# B&R Automation Studio project Software_lab_3
Automation Studio 4.5.2.102

## Logical view

Binary libraries used (declarations not repeated): operator, runtime, astime, AsIecCon, AsBrStr, brsystem, sys_lib, AsIOTime, standard, asstring, Acp10_MC, Acp10man, NcGlobal, Acp10par, Acp10sim, Acp10sdc

### Global.var - Global variables
```iecst
VAR
	Axis_X : ACP10AXIS_typ;
	Axis_X_HW : SdcHwCfg_typ := (0);
	Axis_X_DrvIf : SdcDrvIf16_typ := (0);
	Axis_X_EncIf : SdcEncIf16_typ;
	Axis_X_DiDoIf : SdcDiDoIf_typ := (0);
	Axis_X_ModuleOk : BOOL := 0;
END_VAR
```

### Package Logical/Libraries - Global libraries

### Library Logical/Libraries/MotorCtrl (ANSIC)

#### MotorCtrl.fun - Exported functions and function blocks
```iecst
FUNCTION_BLOCK FB_Regulator
	VAR_INPUT
		e : REAL;
		e_prev : REAL;
	END_VAR
	VAR_OUTPUT
		u : REAL;
	END_VAR
	VAR
		u_raw : REAL;
		k_p : REAL;
		k_i : REAL;
		integrator : FB_Integrator;
		iyOld : REAL;
		max_abs_value : REAL;
	END_VAR
END_FUNCTION_BLOCK

FUNCTION_BLOCK FB_Motor
	VAR_INPUT
		u : REAL;
	END_VAR
	VAR_OUTPUT
		w : REAL;
		phi : REAL;
	END_VAR
	VAR
		integrator : FB_Integrator;
		integrator_phi : FB_Integrator;
		Tm : REAL;
		ke : REAL;
		enable_reg : BOOL;
	END_VAR
END_FUNCTION_BLOCK

FUNCTION_BLOCK FB_Integrator
	VAR_INPUT
		in : REAL;
	END_VAR
	VAR_OUTPUT
		out : REAL;
	END_VAR
	VAR
		dt : REAL;
		direct : BOOL;
	END_VAR
END_FUNCTION_BLOCK

FUNCTION_BLOCK FB_Axis
	VAR_INPUT
		u : USINT;
		endswitch_a_reached : BOOL;
		endswitch_b_reached : BOOL;
	END_VAR
	VAR_OUTPUT
		reset_error : BOOL;
		reset_counter : BOOL;
		pwm_value : INT;
		counter : INT;
		speed : REAL;
	END_VAR
	VAR
		last_counter : INT;
		InMotion : BOOL;
	END_VAR
END_FUNCTION_BLOCK
```

#### FB_Regulator.c
```c
#include <bur/plctypes.h>
#ifdef __cplusplus
	extern "C"
	{
#endif
#include "MotorCtrl.h"
#ifdef __cplusplus
	};
#endif
/* TODO: Add your comment here */
void FB_Regulator(struct FB_Regulator* inst)
{
	if (inst->integrator.direct)
		inst->integrator.in = inst->k_i * inst->e_prev + inst->iyOld / inst->integrator.dt;
	else
		inst->integrator.in = inst->k_i * inst->e + inst->iyOld / inst->integrator.dt;
	FB_Integrator(&inst->integrator);
	inst->u_raw = (inst->k_p * inst->e <= inst->max_abs_value ? inst->k_p * inst->e : inst->max_abs_value) +
		inst->integrator.out;
	inst->u = inst->u_raw < inst->max_abs_value ? inst->u_raw : inst->max_abs_value;
	inst->iyOld = inst->u - inst->u_raw;
}
```

#### FB_Motor.c
```c
#include <bur/plctypes.h>
#ifdef __cplusplus
	extern "C"
	{
#endif
#include "MotorCtrl.h"
#ifdef __cplusplus
	};
#endif
/* TODO: Add your comment here */
void FB_Motor(struct FB_Motor* inst)
{
	inst->integrator.in = (inst->u / inst->ke - inst->w) / inst->Tm;
	FB_Integrator(&inst->integrator);
	inst->w = inst->integrator.out;

	inst->integrator_phi.in = inst->w;
	FB_Integrator(&inst->integrator_phi);
	inst->phi = inst->integrator_phi.out;
}
```

#### FB_Axis.c
```c
#include <bur/plctypes.h>
#ifdef __cplusplus
	extern "C"
	{
#endif
#include "MotorCtrl.h"
#ifdef __cplusplus
	};
#endif
/* TODO: Add your comment here */
void FB_Axis(struct FB_Axis* inst)
{
	if (inst->InMotion)
	{
		if (inst->endswitch_a_reached || inst->endswitch_b_reached)
		{
			inst->pwm_value = 0;
			inst->speed = 0;
			inst->reset_error = 1;
			inst->InMotion = 0;
		}
		else
		{
			inst->pwm_value = inst->u / 24.0 * 32767;
			inst->speed = 50;
			inst->reset_error = 0;
		}
	}
}
```

### Program Logical/SDCAxisCtrlX (ANSIC)

#### Variables.var
```iecst
VAR
	axis_X : FB_Axis;
	coil_powered : BOOL;
	coil_pwm_value : INT;
	fb_regulator : FB_Regulator;
	pwm_period : UINT;
	min_task : INT := 7000;
END_VAR
```

#### Main.c
```c
/*#include <bur/plctypes.h>
#include <math.h>

#ifdef _DEFAULT_INCLUDES
	#include <AsDefault.h>
#endif

#define MOTORS_COUNT 3

void _INIT MainINIT(void)
{
	//Устанавливаем типы SDC модулей
	Axis_X_HW.EncIf1_Typ = ncSDC_ENC16;
	Axis_X_HW.DiDoIf_Typ = ncSDC_DIDO;
	Axis_X_HW.DrvIf_Typ = ncSDC_DRVSERVO16;
	//Устанавливаем имена переменных
	strcpy(Axis_X_HW.EncIf1_Name, "Axis_X_EncIf");
	strcpy(Axis_X_HW.DrvIf_Name, "Axis_X_DrvIf");
	strcpy(Axis_X_HW.DiDoIf_Name, "Axis_X_DiDoIf");
	//Устанавливаем входы готовности и нормальной
	работы
	Axis_X_EncIf.iEncOK = 1;
	Axis_X_DrvIf.iDrvOK = 1;
	Axis_X_DrvIf.iStatusEnable = 1;
	Axis_X_DiDoIf.iDriveReady = 1;

	Axis_X_EncIf.iLifeCnt++;
	Axis_X_DiDoIf.iLifeCntDriveEnable++;
	Axis_X_DiDoIf.iLifeCntDriveReady++;
	Axis_X_DiDoIf.iLifeCntNegHwEnd++;
	Axis_X_DiDoIf.iLifeCntPosHwEnd++;
	Axis_X_DiDoIf.iLifeCntReference++;
	Axis_X_DrvIf.iLifeCnt++;
	Axis_X_EncIf.iActTime = (INT)AsIOTimeCyclicStart();

	int i = 0;
	for (; i < MOTORS_COUNT; i++)
	{
		motors[i].pwm_value = 0;
		motors[i].pwm_percentage = 0;
		motors[i].counter = 0;
		motors[i].coordinate = 0;
		motors[i].button_status = 0;
		motors[i].reset_error = 0;
		motors[i].endswitch_a_reached = 0;
		motors[i].endswitch_b_reached = 0;
	}
	pwm_period = 200;
	coil_powered = 0;
	coil_pwm_value = 0;
	emergency_stop = 0;
	current_motor_index = 0;

	check = 0;
	a = 0;
	n = 0;
}

void _CYCLIC MainCYCLIC(void)
{
	int i = 0, j = 0;
	if (emergency_stop)  //аварийная остановка
	{
		for (i = 0; i < MOTORS_COUNT; i++)
		{
			motors[i].pwm_value = 0;
			motors[i].pwm_percentage = 0;
		}
		coil_powered = 0;
		check = 0;
		emergency_stop = 0;
	}
	current_motor = &motors[current_motor_index];
	for (i = 0; i < MOTORS_COUNT; i++)  //цикл для обозначения на экране текущей степени (кнопка подсвечивается белым цветом)
	{
		MotorFunctionBlock(&motors[i]);
		if (current_motor == &motors[i])
		{
			motors[i].button_status = 1 << 1;
		}
		else
		{
			motors[i].button_status = 0;
		}
	}
	if (coil_powered)  //проверяем напряжение на катушке
	{
		coil_pwm_value = 32767;
		if (check)
		{
			switch (mode)  //проверяем выбранный режим
			{
				case 1:
					switch (path)  //проверяем выбранный контур, разбиваем его и заполняем массив координат соответствующими значениями
					{
						case 1:
							for (i = 0; i < 20; i++)
							{
								coordX[i] = 150 * pi * i / (10*sqrt(2));
								coordY[i] = 150 * pi * i / (10*sqrt(2));
								coordZ[i] = 250 * sin(sqrt(coordX[i] * coordX[i] + coordY[i] * coordY[i]) / 150);
							}
							break;
						case 2:
							for (i = 0; i < 20; i++)
							{
								coordX[i] = 30 * i;
								coordY[i] = 30 * i;
								coordZ[i] = (coordX[i] * coordX[i] + coordY[i] * coordY[i]) / 180;
							}
							break;
						case 0:
							break;
					}
					distX = coordX[a+1] - coordX[a];  //длина полученных отрезков
					distY = coordY[a+1] - coordY[a];
					distZ = coordZ[a+1] - coordZ[a];
					if ((fabs(distX) >= fabs(distY)) && (fabs(distX) >= fabs(distZ)))  //поиск наибольшей проекции каждого отрезка
					{
						index[a] = 2;
					}
					if ((fabs(distY) >= fabs(distX)) && (fabs(distY) >= fabs(distZ)))
					{
						index[a] = 0;
					}
					if ((fabs(distZ) >= fabs(distX)) && (fabs(distZ) >= fabs(distY)))
					{
						index[a] = 1;
					}
					if (index[a] == 2)  //проекция на ось X наибольшая
					{
						if (motors[2].counter > coordX[a+1])  //если степень находится за следующей точкой, то двигаем её в обратном направлении
						{
							motors[2].pwm_percentage_float = -50.0;
						}
						if (motors[2].counter < coordX[a+1])  //если перед точкой, то в прямом направлении
						{
							motors[2].pwm_percentage_float = 50.0;
						}
						motors[0].pwm_percentage_float = (distY * motors[2].pwm_percentage_float) / distX;  //вычисляем реальное значение ШИМ (в процентах)
						motors[1].pwm_percentage_float = (distZ * motors[2].pwm_percentage_float) / distX;
						if ((motors[2].counter >= (coordX[a+1] - 2)) && (motors[2].counter <= (coordX[a+1] + 2)))
						{
							if (a < 18)  //проверка пройденных точек
							{
								a++;
							}
							else  //если все точки пройдены, то отключаем степени и сбрасываем выбранные режим и контур
							{
								for (i = 0; i < MOTORS_COUNT; i++)
								{
									motors[i].pwm_percentage_float = 0.0;
									motors[i].pwm_value_float = 0.0;
									motors[i].pwm_percentage = 0;
									motors[i].pwm_value = 0;
								}
								check = 0;
								mode = 0;
								path = 0;
								a = 0;
							}
						}
					}
					if (index[a] == 0)  //проекция на ось Y максимальная
					{
						if (motors[0].counter > coordY[a+1])  //если степень находится за следующей точкой, то двигаем её в обратном направлении
						{
							motors[0].pwm_percentage_float = -50.0;
						}
						if (motors[0].counter < coordY[a+1])  //если перед точкой, то в прямом направлении
						{
							motors[0].pwm_percentage_float = 50.0;
						}
						motors[2].pwm_percentage_float = (distX * motors[0].pwm_percentage_float) / distY;  //вычисляем реальное значение ШИМ (в процентах)
						motors[1].pwm_percentage_float = (distZ * motors[0].pwm_percentage_float) / distY;
						if ((motors[0].counter >= (coordY[a+1] - 2)) && (motors[0].counter <= (coordY[a+1] + 2)))
						{
							if (a < 18)  //проверка пройденных точек
							{
								a++;
							}
							else  //если все точки пройдены, то отключаем степени и сбрасываем выбранные режим и контур
							{
								for (i = 0; i < MOTORS_COUNT; i++)
								{
									motors[i].pwm_percentage_float = 0.0;
									motors[i].pwm_value_float = 0.0;
									motors[i].pwm_percentage = 0;
									motors[i].pwm_value = 0;
								}
								check = 0;
								mode = 0;
								path = 0;
								a = 0;
							}
						}
					}
					if (index[a] == 1)  //проекция на ось Z максимальная
					{
						if (motors[1].counter > coordZ[a+1])  //если степень находится за следующей точкой, то двигаем её в обратном направлении
						{
							motors[1].pwm_percentage_float = -50.0;
						}
						if (motors[1].counter < coordZ[a+1])  //если перед точкой, то в прямом направлении
						{
							motors[1].pwm_percentage_float = 50.0;
						}
						motors[2].pwm_percentage_float = (distX * motors[1].pwm_percentage_float) / distZ;  //вычисляем реальное значение ШИМ (в процентах)
						motors[0].pwm_percentage_float = (distY * motors[1].pwm_percentage_float) / distZ;
						if ((motors[1].counter >= (coordZ[a+1] - 2)) && (motors[1].counter <= (coordZ[a+1] + 2)))
						{
							if (a < 18)  //проверка пройденных точек
							{
								a++;
							}
							else  //если все точки пройдены, то отключаем степени и сбрасываем выбранные режим и контур
							{
								for (i = 0; i < MOTORS_COUNT; i++)
								{
									motors[i].pwm_percentage_float = 0.0;
									motors[i].pwm_value_float = 0.0;
									motors[i].pwm_percentage = 0;
									motors[i].pwm_value = 0;
								}
								check = 0;
								mode = 0;
								path = 0;
								a = 0;
							}
						}
					}
					for (i = 0; i < MOTORS_COUNT; i++)
					{
						motors[i].pwm_percentage = motors[i].pwm_percentage_float;  //присваиваем значению ШИМ на слайдере на экране к реальному значению ШИМ (для наглядности)
					}
					for (i = 0; i < MOTORS_COUNT; i++)
					{
						motors[i].pwm_value_float = 32767 * motors[i].pwm_percentage_float / 100;  //вычисляем ШИМ для каждой степени
						motors[i].pwm_value = motors[i].pwm_value_float;  //приводим значение типа REAL к значению типа INT и пересылаем на двигатель
						if ((!motors[i].endswitch_a_reached) && (!motors[i].endswitch_b_reached))
						{
							motors[i].reset_error = 0;
						}
						if ((motors[i].endswitch_a_reached) && (motors[i].pwm_percentage > 0))  //если достигнут концевой датчик, то останавливаем все степени и сбрасываем ошибку
						{
							motors[i].reset_error = 1;
							for (j = 0; j < MOTORS_COUNT; j++)
							{
								motors[j].pwm_percentage_float = 0.0;
								motors[j].pwm_value_float = 0.0;
								motors[j].pwm_percentage = 0;
								motors[j].pwm_value = 0;
							}
						}
						if ((motors[i].endswitch_b_reached) && (motors[i].pwm_percentage < 0))
						{
							motors[i].reset_error = 1;
							for (j = 0; j < MOTORS_COUNT; j++)
							{
								motors[j].pwm_percentage_float = 0.0;
								motors[j].pwm_value_float = 0.0;
								motors[j].pwm_percentage = 0;
								motors[j].pwm_value = 0;
							}
						}
					}
					break;  //закрытие 1-го режима
				case 2:
					switch (path)  //проверяем выбранный контур и задаем соответствующие функции изменения скоростей движения степеней
					{
						case 1:
							motors[0].pwm_percentage_float = 50.0;
							motors[2].pwm_percentage_float = 50.0;
							motors[1].pwm_percentage_float = 90 * cos(pi * n / 40);
							break;
						case 2:
							motors[0].pwm_percentage_float = 50.0;
							motors[2].pwm_percentage_float = 50.0;
							if ((n * n / 60) <= 100)  //ШИМ не может быть больше 100%
							{
								motors[1].pwm_percentage_float = n * n / 60;
							}
							else  //если больше 100%, то отключаем степени и сбрасываем выбранные режим и контур
							{
								for (i = 0; i < MOTORS_COUNT; i++)
								{
									motors[i].pwm_percentage_float = 0.0;
									motors[i].pwm_value_float = 0.0;
									motors[i].pwm_percentage = 0;
									motors[i].pwm_value = 0;
								}
								check = 0;
								mode = 0;
								path = 0;
								n = 0;
							}
						case 0:
							break;
					}
					if (n < 80)  //за 1 секунду проходит 10 итераций основного цикла; если движение происходит 8 секунд, то к концу 8-ой секунды пройдет 80 итераций
					{
					n++;
					}
					else  //если все итерации пройдены, то отключаем степени и сбрасываем выбранные режим и контур
					{
					for (i = 0; i < MOTORS_COUNT; i++)
					{
					motors[i].pwm_percentage_float = 0.0;
					motors[i].pwm_value_float = 0.0;
					motors[i].pwm_percentage = 0;
					motors[i].pwm_value = 0;
					}
					check = 0;
					mode = 0;
					path = 0;
					n = 0;
					}
					for (i = 0; i < MOTORS_COUNT; i++)
					{
						motors[i].pwm_percentage = motors[i].pwm_percentage_float;  //присваиваем значению ШИМ на слайдере на экране к реальному значению ШИМ (для наглядности)
					}
					for (i = 0; i < MOTORS_COUNT; i++)
					{
						motors[i].pwm_value_float = 32767 * motors[i].pwm_percentage_float / 100;  //вычисляем ШИМ для каждой степени
						motors[i].pwm_value = motors[i].pwm_value_float;  //приводим значение типа REAL к значению типа INT и пересылаем на двигатель
						if ((!motors[i].endswitch_a_reached) && (!motors[i].endswitch_b_reached))
						{
							motors[i].reset_error = 0;
						}
						if ((motors[i].endswitch_a_reached) && (motors[i].pwm_percentage > 0))  //если достигнут концевой датчик, то останавливаем все степени и сбрасываем ошибку
						{
							motors[i].reset_error = 1;
							for (j = 0; j < MOTORS_COUNT; j++)
							{
								motors[j].pwm_percentage_float = 0.0;
								motors[j].pwm_value_float = 0.0;
								motors[j].pwm_percentage = 0;
								motors[j].pwm_value = 0;
							}
						}
						if ((motors[i].endswitch_b_reached) && (motors[i].pwm_percentage < 0))
						{
							motors[i].reset_error = 1;
							for (j = 0; j < MOTORS_COUNT; j++)
							{
								motors[j].pwm_percentage_float = 0.0;
								motors[j].pwm_value_float = 0.0;
								motors[j].pwm_percentage = 0;
								motors[j].pwm_value = 0;
							}
						}
					}
					break;  //закрытие 2-го режима
				case 0:
					break;
			}
		}
		else  //если движение не начато, то переходим в режим ручного управления через сенсорный экран (для отладки, приведения в начало координат и т.д.)
		{
			for (i = 0; i < MOTORS_COUNT; i++)
			{
				motors[i].pwm_value = 32767 * motors[i].pwm_percentage / 100;
				if ((!motors[i].endswitch_a_reached) && (!motors[i].endswitch_b_reached))
				{
					motors[i].reset_error = 0;
				}
				if ((motors[i].endswitch_a_reached) && (motors[i].pwm_percentage > 0))
				{
					motors[i].reset_error = 1;
					motors[i].pwm_percentage = 0;
					motors[i].pwm_value = 0;
				}
				if ((motors[i].endswitch_b_reached) && (motors[i].pwm_percentage < 0))
				{
					motors[i].reset_error = 1;
					motors[i].pwm_percentage = 0;
					motors[i].pwm_value = 0;
				}
			}
		}
	}
	else  //если нет напряжения на катушке, то отключаем все степени
	{
		coil_pwm_value = 0;
		for (i = 0; i < MOTORS_COUNT; i++)
		{
			motors[i].pwm_value = 0;
		}
	}
}

void _EXIT ProgramExit(void)
{

}*/

#include <bur/plctypes.h>
#include <standard.h>
#include <string.h>
#include <bur/plc.h>
#ifdef _DEFAULT_INCLUDES
#include <AsDefault.h>

#endif

void increase_counters(void);

void _INIT ProgramInit(void)
{
	//Устанваливаем типы SDC модулей
	Axis_X_HW.EncIf1_Typ = ncSDC_ENC16;
	Axis_X_HW.DiDoIf_Typ = ncSDC_DIDO;
	Axis_X_HW.DrvIf_Typ = ncSDC_DRVSERVO16;

	//Устанавливаем имена переменных
	strcpy(Axis_X_HW.EncIf1_Name, "Axis_X_EncIf");
	strcpy(Axis_X_HW.DrvIf_Name, "Axis_X_DrvIf");
	strcpy(Axis_X_HW.DiDoIf_Name, "Axis_X_DiDoIf");

	//Устанавливаем входы готовности и нормальной работы
	Axis_X_EncIf.iEncOK = 1;
	Axis_X_DrvIf.iDrvOK = 1;
	Axis_X_DrvIf.iStatusEnable = 1;
	Axis_X_DiDoIf.iDriveReady = 1;

	fb_regulator.integrator.dt = 0.002;
	fb_regulator.k_i = 0.16 * 0.01;
	fb_regulator.k_p = 0.0064 * 0.01;
	fb_regulator.max_abs_value = 24.0;

	pwm_period = 200;

	axis_X.InMotion = 1;
}

void _CYCLIC ProgramCyclic(void)
{
	increase_counters();
	Axis_X_EncIf.iActTime = (INT)	AsIOTimeCyclicStart();

	Axis_X_EncIf.iActPos = axis_X.counter++;
	Axis_X_DiDoIf.iPosHwEnd = axis_X.endswitch_b_reached;
	Axis_X_DiDoIf.iNegHwEnd = axis_X.endswitch_a_reached;

	if (coil_powered)
	{
		coil_pwm_value = 32767;

		//fb_regulator.e = Axis_X_DrvIf.oSetPos * 6500 / 32767 - axis_X.speed * 100;
		//FB_Regulator(&fb_regulator);

		axis_X.u = 18;  //fb_regulator.u
		FB_Axis(&axis_X);
	}
}

void increase_counters(void)
{
	Axis_X_EncIf.iLifeCnt++;
	Axis_X_DiDoIf.iLifeCntDriveEnable++;
	Axis_X_DiDoIf.iLifeCntDriveReady++;
	Axis_X_DiDoIf.iLifeCntNegHwEnd++;
	Axis_X_DiDoIf.iLifeCntPosHwEnd++;
	Axis_X_DiDoIf.iLifeCntReference++;
	Axis_X_DrvIf.iLifeCnt++;
}

void _EXIT ProgramExit(void)
{
	// Insert code here

}
```

### Program Logical/ncsdcctrl (IEC)

#### ncsdcctrl.var
```iecst
VAR
	Axis_X_oSetPosOld : INT := 0;
END_VAR
```

#### ncsdcctrlCyclic.st
```iecst
PROGRAM _CYCLIC

(* ### BEGIN Axis_X ### *)

(* life counter emulation of digital inputs *)
        Axis_X_DiDoIf.iLifeCntReference := Axis_X_DiDoIf.iLifeCntReference + 1;
        Axis_X_DiDoIf.iLifeCntNegHwEnd  := Axis_X_DiDoIf.iLifeCntNegHwEnd  + 1;
        Axis_X_DiDoIf.iLifeCntPosHwEnd  := Axis_X_DiDoIf.iLifeCntPosHwEnd  + 1;

(* ### END Axis_X ### *)

END_PROGRAM
```

#### ncsdcctrlInit.st
```iecst
PROGRAM _INIT

(* ### BEGIN Axis_X ### *)

(* initialize variables *)
        Axis_X_HW.DrvIf_Typ := ncSDC_DRVSERVO16;
        brsstrcpy(ADR(Axis_X_HW.DrvIf_Name[0]), ADR('Axis_X_DrvIf'));
        Axis_X_HW.DiDoIf_Typ := ncSDC_DIDO;
        brsstrcpy(ADR(Axis_X_HW.DiDoIf_Name[0]), ADR('Axis_X_DiDoIf'));

(* force variable offset generation *)
        Axis_X.size                      := Axis_X.size;
        Axis_X_DrvIf.iLifeCnt            := Axis_X_DrvIf.iLifeCnt;
        Axis_X_DiDoIf.iLifeCntDriveReady := Axis_X_DiDoIf.iLifeCntDriveReady;
        Axis_X_ModuleOk                  := Axis_X_ModuleOk;

(* assign your hardware inputs here*)

(*      Axis_X_DiDoIf.iPosHwEnd  := Axis_X_DiDoIf.iPosHwEnd;
        Axis_X_DiDoIf.iNegHwEnd  := Axis_X_DiDoIf.iNegHwEnd;
        Axis_X_DiDoIf.iReference := Axis_X_DiDoIf.iReference;
 *)

(* ### END Axis_X ### *)

END_PROGRAM
```

### Package Logical/Axis_Xobj - gAxis02obj

### Data object Logical/Axis_Xobj/Axis_Xa (Apt)

#### Axis_Xa.apt
```
AcoposParameterTable:
  Root Parameters:
    230 = PCTRL_S_SET (Name=PCTRL_S_ACT_PARID)
    64201 = 6500 (Name=SERVO_V_MAX_OUTPUT)
```

### Data object Logical/Axis_Xobj/Axis_Xi (Ax)

#### Axis_Xi.ax
```
InitParameter (Version=5.02.1, NcSwId=Acp10)
  ACP10AXIS_typ:
    dig_in:
      level:
        reference = ncACTIV_HI
        pos_hw_end = ncACTIV_HI
        neg_hw_end = ncACTIV_HI
        trigger1 = ncACTIV_HI
        trigger2 = ncACTIV_LO + ncQUICKSTOP
    encoder_if:
      parameter:
        count_dir = ncSTANDARD
        scaling:
          load:
            units = 3000
            rev_motor = 1
    limit:
      parameter:
        v_pos = 10000
        v_neg = 10000
        a1_pos = 10000.0
        a2_pos = 10000.0
        a1_neg = 10000.0
        a2_neg = 10000.0
        t_jolt = 0
        t_in_pos = 0
        pos_sw_end = 2000000000
        neg_sw_end = -2000000000
        ds_warning = 500
        ds_stop = 50000.0
        a_stop = 1.0e30
        dv_stop = 0
        dv_stop_mode = ncOFF
    controller:
      mode = ncPOSITION
      position:
        kv = 50
        tn = 0
        t_predict = 0.01
        t_total = 0.01
        p_max = 1.0e30
        i_max = 0
      speed:
        kv = 2.0
        tn = 0
        t_filter = 0.0
        isq_filter1:
          type = ncOFF
          a0 = 0.0
          a1 = 0.0
          b0 = 0.0
          b1 = 0.0
          b2 = 0.0
          c0_par_id = 0
          c1_par_id = 0
        isq_filter2:
          type = ncOFF
          a0 = 0.0
          a1 = 0.0
          b0 = 0.0
          b1 = 0.0
          b2 = 0.0
          c0_par_id = 0
          c1_par_id = 0
        isq_filter3:
          type = ncOFF
          a0 = 0.0
          a1 = 0.0
          b0 = 0.0
          b1 = 0.0
          b2 = 0.0
          c0_par_id = 0
          c1_par_id = 0
      uf:
        type = ncLINEAR + ncCORRECTION
        auto_config = ncMOTOR_PAR
        u0 = 0
        un = 0
        fn = 50.0
        k_f_slip = 0
      ff:
        torque_load = 0.0
        torque_pos = 0.0
        torque_neg = 0.0
        kv_torque = 0.0
        inertia = 0.0
        t_filter_a = 0.0
    move:
      stop:
        parameter[0]:
          decel_ramp = ncA_LIMIT
          controller = ncON
        parameter[1]:
          decel_ramp = ncA_LIMIT
          controller = ncON
        parameter[2]:
          decel_ramp = ncA_LIMIT
          controller = ncON
        parameter[3]:
          decel_ramp = ncA_LIMIT
          controller = ncON
        quickstop:
          decel_ramp = ncA_LIMIT
          t_jolt = 0
        drive_error:
          decel_ramp = ncA_LIMIT
      homing:
        parameter:
          s = 0
          v_switch = 6000.0
          v_trigger = 2000.0
          a = 10000.0
          mode = ncEND_SWITCH
          edge_sw = ncNEGATIVE
          start_dir = ncPOSITIVE
          trigg_dir = ncNEGATIVE
          ref_pulse = ncOFF
          fix_dir = ncOFF
          tr_s_block = 0
          torque_lim = 0
          ds_block = 0
          ds_stop = 0
      basis:
        parameter:
          v_pos = 5000
          v_neg = 5000
          a1_pos = 50000
          a2_pos = 50000
          a1_neg = 50000
          a2_neg = 50000
    message:
      text:
        parameter:
          format = ncBREAK
          columns = 80
          data_modul = acp10etxen
```

Listed in the project but not available here: Logical/Global.typ, Logical/Libraries/MotorCtrl/Types.typ, Logical/Libraries/MotorCtrl/Constants.var, Logical/Libraries/MotorCtrl/FB_Integrator.c, Logical/acp10etxen
